Omron Sysmac Studio project NilsTestProject (Sysmac Studio 1.18.0.15, StandardProject)
(* Just a test program *)

# Controller new_Controller_0: NJ101-9000 version 1.13
Units and slaves: Power Supply : NJ-Px3001; CPU : NJ101-9000; 0 : CJ1W-ID211 (J01); 1 : CJ1W-OD212 (J02); 2 [Unit 0] : CJ1W-AD041-V1 (J03)
Task PrimaryTask (priority 4, period or condition 2000): TraficLightSfc

TYPE SFC : (STEP01 := 0 (* Step 1 *), STEP02 := 1 (* Step 2 *)); END_TYPE

VAR_GLOBAL
    iTl1GreenReqBtn : BOOL;  (* Trafic Light 1: Green request button (100S1); at IOBus://rack#0/slot#0/Ch1_In/Ch1_In00 *)
    iTl2GreenReqBtn : BOOL;  (* Trafic Light 2: Green request button (100S2); at IOBus://rack#0/slot#0/Ch1_In/Ch1_In01 *)
    oTl1RedLgt : BOOL;  (* Trafic Light 1: Red light (110H1); at IOBus://rack#0/slot#1/Ch1_Out/Ch1_Out00 *)
    oTl1OrangeLgt : BOOL;  (* Trafic Light 1: Orange light (110H2); at IOBus://rack#0/slot#1/Ch1_Out/Ch1_Out01 *)
    oTl1GreenLgt : BOOL;  (* Trafic Light 1: Green light (110H3); at IOBus://rack#0/slot#1/Ch1_Out/Ch1_Out02 *)
    oTl2RedLgt : BOOL;  (* Trafic Light 2: Red light (111H1); at IOBus://rack#0/slot#1/Ch1_Out/Ch1_Out03 *)
    oTl2OrangeLgt : BOOL;  (* Trafic Light 2: Orange light (111H2); at IOBus://rack#0/slot#1/Ch1_Out/Ch1_Out04 *)
    oTl2GreenLgt : BOOL;  (* Trafic Light 2: Green light (111H3); at IOBus://rack#0/slot#1/Ch1_Out/Ch1_Out05 *)
    iTest1 : BOOL;  (* Test input 1; at IOBus://rack#0/slot#0/Ch1_In/Ch1_In03 *)
    iTest2 : BOOL;  (* Test input 2; at IOBus://rack#0/slot#0/Ch1_In/Ch1_In04 *)
END_VAR

PROGRAM TraficLightSfc
VAR
    T_Tl1OTl2O : BOOL;  (* Trafic light 1: Orange, Trafic light 2: Orange *)
    T_Tl1RTl2R : BOOL;  (* Trafic light 1: Red, Trafic light 2: Red *)
    T_Tl1GTl2R : BOOL;  (* Trafic light 1: Green Trafic light 2: Red *)
    F_KeepTl1OTl2O : SR;
    OrangeDelay : _sTimer;
    Test : BOOL;  (* This is symbol 1 *)
    Test1 : BOOL;
END_VAR
VAR_EXTERNAL
    I_Tl1GreenReqBtn : BOOL;
    O_Tl1GreenLgt : BOOL;
END_VAR
VAR
    _t1 : BOOL;
END_VAR

(* Section Section0: ladder, written here as Structured Text *)

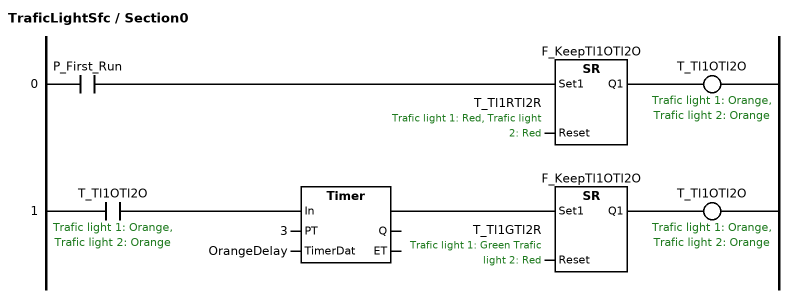
(* Rung 0 *)
F_KeepTl1OTl2O(Set1 := P_First_Run, Reset := T_Tl1RTl2R);
T_Tl1OTl2O := F_KeepTl1OTl2O.Q1;
(* Rung 1 *)
_t1 := Timer(In := T_Tl1OTl2O, PT := 3, TimerDat := OrangeDelay);
F_KeepTl1OTl2O(Set1 := _t1, Reset := T_Tl1GTl2R);
T_Tl1OTl2O := F_KeepTl1OTl2O.Q1;
END_PROGRAM

PROGRAM SfcTest
VAR
    Sfc : INT;  (* Sequential Flow Chart: Actual step nr *)
END_VAR

(* Section Sfc: ladder, written here as Structured Text *)

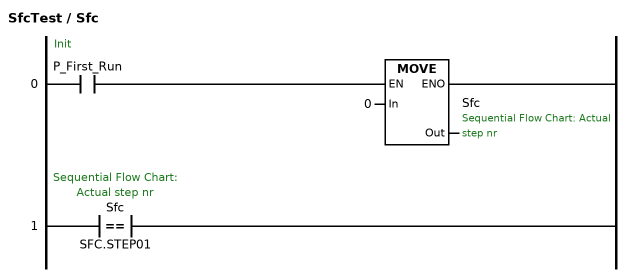
(* Rung 0: Init *)
IF P_First_Run THEN Sfc := 0; END_IF;
(* Rung 1 *)
(* drawn but driving nothing: Sfc, SFC.STEP01 *)
END_PROGRAM

PROGRAM SimpleThings
VAR
    iTest1 : BOOL;  (* Input variable 1 *)
    iTest2 : BOOL;  (* Input Variable 2 *)
    oTest1 : BOOL;  (* Ouput variabale 1 *)
    oTest2 : BOOL;  (* Output variable 2 *)
    oTest3 : BOOL;  (* Output variable 3 *)
    fOnDelay : TON;  (* On Delay *)
    sOnDelayRemTim : TIME;  (* On delay remaining time *)
END_VAR
VAR
    _e1 : R_TRIG;
END_VAR

(* Section SimpleThings: ladder, written here as Structured Text *)

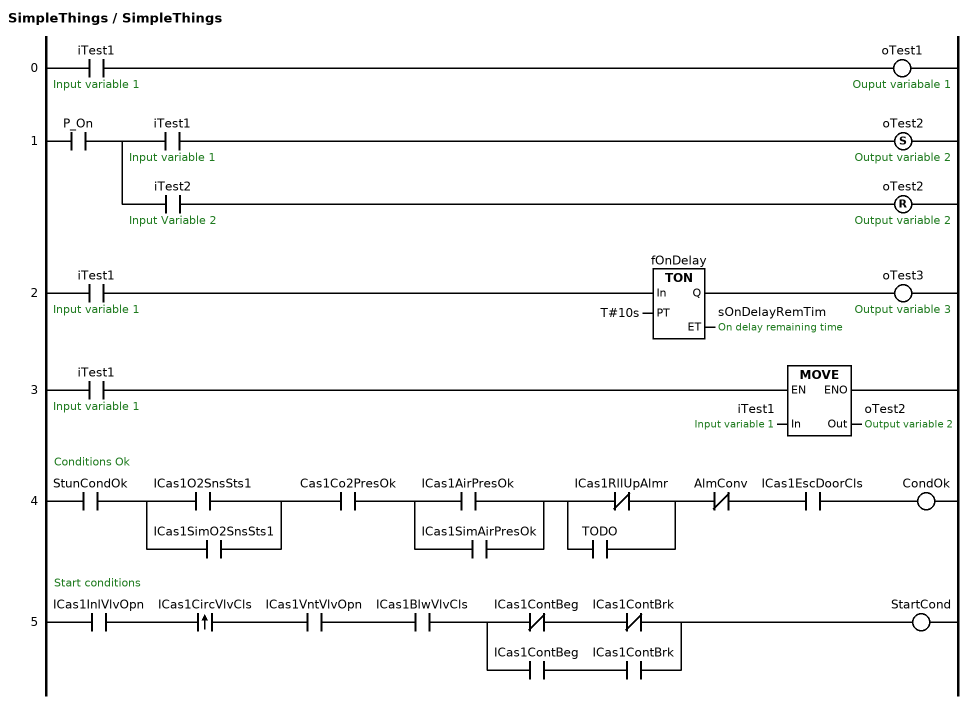
(* Rung 0 *)
oTest1 := iTest1;
(* Rung 1 *)
IF P_On AND iTest1 THEN oTest2 := TRUE; END_IF;
IF P_On AND iTest2 THEN oTest2 := FALSE; END_IF;
(* Rung 2 *)
fOnDelay(In := iTest1, PT := T#10s, ET => sOnDelayRemTim);
oTest3 := fOnDelay.Q;
(* Rung 3 *)
IF iTest1 THEN oTest2 := iTest1; END_IF;
(* Rung 4: Conditions Ok *)
CondOk := StunCondOk AND (ICas1O2SnsSts1 OR ICas1SimO2SnsSts1) AND Cas1Co2PresOk AND (ICas1AirPresOk OR ICas1SimAirPresOk) AND (NOT ICas1RllUpAlmr OR TODO) AND NOT AlmConv AND ICas1EscDoorCls;
(* Rung 5: Start conditions *)
_e1(CLK := ICas1CircVlvCls);
StartCond := ICas1InlVlvOpn AND _e1.Q AND ICas1VntVlvOpn AND ICas1BlwVlvCls AND ((NOT ICas1ContBeg AND NOT ICas1ContBrk) OR (ICas1ContBeg AND ICas1ContBrk));
END_PROGRAM

# Device HMI_NA5_0 (NA): not converted